{attribute 'qualified_only'}
VAR_GLOBAL
		ECAT_x : ECAT_x_A7FD7D81;
END_VAR

(* stored: Version 1.2.0.0, ProductVersion 3.1.4024.12
   GVL GVL_iXlinker: Id {30981106-2311-061b-0048-d4afdaef963f} *)
